SUBAPPLICATION OPC_SUB_EX_1 (* Subapplication Type *)
  (* Standard: 61499-2 *)
  (* Version 1.0, 2022-03-09, Maximilian Scharf *)
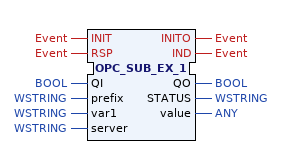
  EVENT_INPUT
    INIT;
    RSP;
  END_EVENT
  EVENT_OUTPUT
    INITO;
    IND;
  END_EVENT
  VAR_INPUT
    QI : BOOL;
    prefix : WSTRING;
    var1 : WSTRING;
    server : WSTRING;
  END_VAR
  VAR_OUTPUT
    QO : BOOL;
    STATUS : WSTRING;
    value : ANY;
  END_VAR
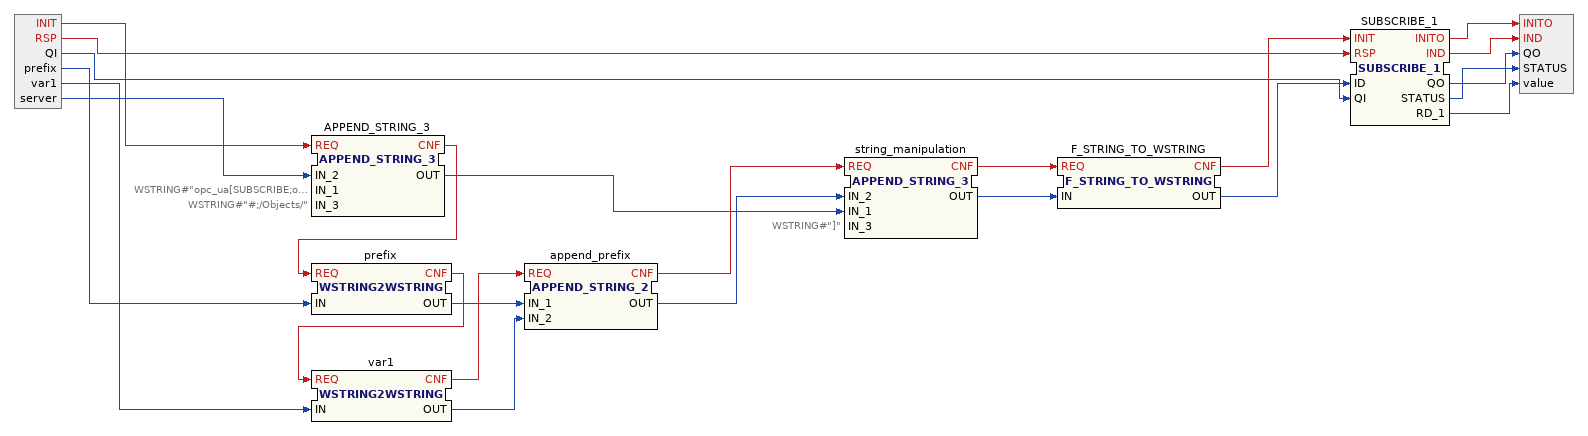
  (* Group __Group01: Example: &#10;SUBSCRIBE &#10;&quot;opc_ua[READ;opc.tcp://localhost:4840#;/Objects/test2]&quot; *)
  FBS
    F_STRING_TO_WSTRING : F_STRING_TO_WSTRING;
    string_manipulation : APPEND_STRING_3(IN_3 := WSTRING#"]");
    var1 : WSTRING2WSTRING;
    SUBSCRIBE_1 : SUBSCRIBE_1;
    append_prefix : APPEND_STRING_2;
    prefix : WSTRING2WSTRING;
    APPEND_STRING_3 : APPEND_STRING_3(IN_1 := WSTRING#"opc_ua[SUBSCRIBE;opc.tcp://", IN_3 := WSTRING#"#;/Objects/");
  END_FBS
  EVENT_CONNECTIONS
    string_manipulation.CNF TO F_STRING_TO_WSTRING.REQ;
    F_STRING_TO_WSTRING.CNF TO SUBSCRIBE_1.INIT;
    SUBSCRIBE_1.INITO TO INITO;
    RSP TO SUBSCRIBE_1.RSP;
    SUBSCRIBE_1.IND TO IND;
    prefix.CNF TO var1.REQ;
    var1.CNF TO append_prefix.REQ;
    INIT TO APPEND_STRING_3.REQ;
    APPEND_STRING_3.CNF TO prefix.REQ;
    append_prefix.CNF TO string_manipulation.REQ;
  END_CONNECTIONS
  DATA_CONNECTIONS
    string_manipulation.OUT TO F_STRING_TO_WSTRING.IN;
    var1 TO var1.IN;
    F_STRING_TO_WSTRING.OUT TO SUBSCRIBE_1.ID;
    SUBSCRIBE_1.QO TO QO;
    SUBSCRIBE_1.STATUS TO STATUS;
    SUBSCRIBE_1.RD_1 TO value;
    QI TO SUBSCRIBE_1.QI;
    prefix TO prefix.IN;
    prefix.OUT TO append_prefix.IN_1;
    var1.OUT TO append_prefix.IN_2;
    append_prefix.OUT TO string_manipulation.IN_2;
    server TO APPEND_STRING_3.IN_2;
    APPEND_STRING_3.OUT TO string_manipulation.IN_1;
  END_CONNECTIONS
END_SUBAPPLICATION
